ABB RobotStudio station: Components.rspag

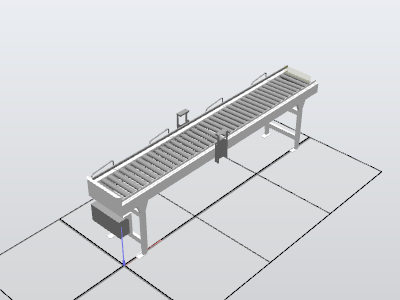
Station Station (saved by RobotStudio 22.3.10190.2)
Layout (positions relative to the parent item):
  - Red_box [part] at (0, 300, 0) mm, size 100 x 100 x 100 mm
  - Green_box [part] at (0, 150, 0) mm, size 100 x 100 x 100 mm
  - Blue_box [part], size 100 x 100 x 100 mm
  - Conveyor [smart component, from Libraries\Conveyor.rslib]
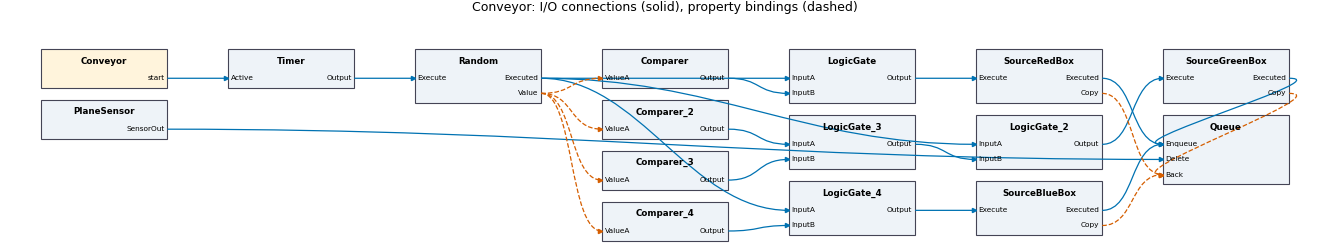
      connections:
        Conveyor.start -> Timer.Active
        Timer.Output -> Random.Execute
        Random.Executed -> LogicGate.InputA
        Comparer.Output -> LogicGate.InputB
        Random.Executed -> LogicGate_2.InputA
        Comparer_2.Output -> LogicGate_3.InputA
        Comparer_3.Output -> LogicGate_3.InputB
        LogicGate_3.Output -> LogicGate_2.InputB
        Random.Executed -> LogicGate_4.InputA
        Comparer_4.Output -> LogicGate_4.InputB
        LogicGate.Output -> SourceRedBox.Execute
        LogicGate_2.Output -> SourceGreenBox.Execute
        LogicGate_4.Output -> SourceBlueBox.Execute
        SourceRedBox.Executed -> Queue.Enqueue
        SourceGreenBox.Executed -> Queue.Enqueue
        SourceBlueBox.Executed -> Queue.Enqueue
        PlaneSensor.SensorOut -> Queue.Delete
        Random.Value => Comparer.ValueA
        Random.Value => Comparer_2.ValueA
        Random.Value => Comparer_3.ValueA
        Random.Value => Comparer_4.ValueA
        SourceRedBox.Copy => Queue.Back
        SourceGreenBox.Copy => Queue.Back
        SourceBlueBox.Copy => Queue.Back
    - SourceRedBox [smart component, from Components\Source.rslib]
        properties: Source=Red_box; Copy=(none); Parent=(none); Position=[0.075 0.17 0.775]; Orientation=[0 0 0]; Transient=true; PhysicsBehavior=-1
    - SourceGreenBox [smart component, from Components\Source.rslib]
        properties: Source=Green_box; Copy=(none); Parent=(none); Position=[0.075 0.17 0.775]; Orientation=[0 0 0]; Transient=true; PhysicsBehavior=-1
    - SourceBlueBox [smart component, from Components\Source.rslib]
        properties: Source=Blue_box; Copy=(none); Parent=(none); Position=[0.075 0.17 0.775]; Orientation=[0 0 0]; Transient=true; PhysicsBehavior=-1
    - Random [smart component, from Components\Random.rslib]
        properties: Value=2.60545295877636; Min=0; Max=3
    - Comparer [smart component, from Components\Comparer.rslib]
        properties: ValueA=2.60545295877636; Operator=<=; ValueB=1
    - Timer [smart component, from Components\Timer.rslib]
        properties: StartTime=0; Interval=3; Repeat=true; CurrentTime=62.472
    - Comparer_2 [smart component, from Components\Comparer.rslib]
        properties: ValueA=2.60545295877636; Operator=>; ValueB=1
    - Comparer_3 [smart component, from Components\Comparer.rslib]
        properties: ValueA=2.60545295877636; Operator=<=; ValueB=2
    - LogicGate [smart component, from Components\LogicGate.rslib]
        properties: Operator=AND; Delay=0
    - LogicGate_2 [smart component, from Components\LogicGate.rslib]
        properties: Operator=AND; Delay=0
    - LogicGate_3 [smart component, from Components\LogicGate.rslib]
        properties: Operator=AND; Delay=0
    - LogicGate_4 [smart component, from Components\LogicGate.rslib]
        properties: Operator=AND; Delay=0
    - Comparer_4 [smart component, from Components\Comparer.rslib]
        properties: ValueA=2.60545295877636; Operator=>; ValueB=2
    - Queue [smart component, from Components\Queue.rslib]
        properties: Back=(none); Front=(none); Queue={ad5028a6-b78d-4c1e-932c-58387a76d111};{caccf65a-5e8a-4d59-86cf-dea641d388fc};{d5145b48-5921-41e5-a5cf-f289e25e2c56};{eb20e8fc-2243-4132-bafd-30e74f28caf8};{df543072-238f-4cf0-af28-d52d1ae9a375};{1c01fbfb-bd7a-479c-aabf-7e294c76dd45};{cb4fb4ea-8899-44f1-8836-deb4a8ef6429};{4a7ed11f-3483-4d0f-abfe-d523fadb1b42};{0f8e3dc3-db70-4297-9f91-4c7c364b3beb};{c87a5a8a-da50-415a-a569-0345de37618b};{a8b1a2bd-e0b2-4c05-9cb6-234d8fd6809a}; NumberOfObjects=9
    - LinearMover [smart component, from Components\LinearMover.rslib]
        properties: Object=Queue; Direction=[1 0 0]; Speed=0.1; Reference=Global; ReferenceObject=(none)
    - PlaneSensor [smart component, from Components\PlaneSensor.rslib]
        properties: Origin=[2.910135 0.39 0.78]; Axis1=[0 -0.38 0]; Axis2=[0 0 0.1]; Tag=(none); SensedPart=(none)
      - _sensorPart_ [part, from Libraries\Conveyor.rslib]
    - 400_guide [part, from Libraries\Conveyor.rslib]
